FUNCTION_BLOCK LWordPointerComparer EXTENDS Object IMPLEMENTS IPointerComparer
VAR
	_ClassName : STRING := __POUNAME();
END_VAR

{attribute 'monitoring' := 'call'}
PROPERTY ClassName : STRING
GET
ClassName := _ClassName;
END_GET
END_PROPERTY

{attribute "object_name" := "Compare"}
METHOD Compare : COMPARISION_RESULT
VAR_INPUT
	left : PVOID;
	right : PVOID;
END_VAR
VAR
	leftPointer : POINTER TO LWORD; 
	rightPointer : POINTER TO LWORD; 
END_VAR
IF left = 0 AND right = 0 THEN
	Compare := COMPARISION_RESULT.FIRST_EQUAL_TO_SECOND;
	RETURN;
END_IF

IF left = 0 THEN
	Compare := COMPARISION_RESULT.FIRST_LESS_THAN_SECOND;
	RETURN;	
END_IF

IF right = 0 THEN
	Compare := COMPARISION_RESULT.FIRST_GREATER_THAN_SECOND;
	RETURN;	
END_IF

leftPointer := left;
rightPointer := right;

IF leftPointer^ < rightPointer^ THEN
	Compare := COMPARISION_RESULT.FIRST_LESS_THAN_SECOND;
ELSIF leftPointer^ > rightPointer^ THEN
	Compare := COMPARISION_RESULT.FIRST_GREATER_THAN_SECOND;
ELSE
	Compare := COMPARISION_RESULT.FIRST_EQUAL_TO_SECOND;	
END_IF
END_METHOD

{attribute 'monitoring' := 'call'}
PROPERTY Size : ULINT
GET
Size := XSIZEOF(THIS^);
END_GET
END_PROPERTY

END_FUNCTION_BLOCK

(* stored: Version 1.1.0.1
   POU LWordPointerComparer: Id {44dfb5c1-f87c-44fd-9232-8e844ccb3ec9}, SpecialFunc None
   Property ClassName: Id {415841df-04fa-491b-a4b5-f850745ee63d}
   Get Get: Id {9ac0da90-0661-440b-a428-9249215adcfb}
   Method Compare: Id {e1d57163-1956-4347-bc1f-49374e441b81}
   Property Size: Id {c20779ba-54df-4c3e-ada4-9b22ccc2cce2}
   Get Get: Id {58eb9c35-923e-4069-bab1-ad5b71fb1a41} *)
